{attribute addProperty BoxType "EJ2918-0000-0017"}
{attribute addProperty Id "FSoE_InputsFSoE_Inputs_3EC5F4AF486FSoE_OutputsFSoE_Outputs_66F1C5B7567"}
{attribute addProperty CRC "4235450693"}
{attribute addProperty SizeInBites "104"}
{attribute addProperty SizeInBytes "13"}
TYPE Module_1_FSOE_FC73D945 :
STRUCT
	{attribute addProperty Name "FSoE_Inputs"}
	FSoE_Inputs  : FSoE_Inputs_3EC5F4AF;
	{attribute addProperty Name "FSoE_Outputs"}
	FSoE_Outputs  : FSoE_Outputs_66F1C5B7;
END_STRUCT
END_TYPE

(* stored: Version 1.2.0.0, ProductVersion 3.1.4024.9
   DUT Module_1_FSOE_FC73D945: Id {bcfe5855-498f-471d-b18b-7271c8291d8d} *)
